FUNCTION_BLOCK C_BINARYREADER
VAR_INPUT
END_VAR
VAR_OUTPUT
END_VAR
VAR
	_BASESTREAM 	: I_STREAM;
END_VAR

PROPERTY BaseStream : I_STREAM
GET
BaseStream := _BASESTREAM;
END_GET
END_PROPERTY

METHOD Close : DINT
VAR_INPUT
END_VAR
Close := _BASESTREAM.Close();
_BASESTREAM := 0;
RETURN;
END_METHOD

METHOD New : DINT
VAR_INPUT
	STREAM : I_STREAM;
END_VAR
IF STREAM = 0 THEN
	New := 1;
	RETURN;
ELSE
	IF STREAM.IsValid THEN
		_BASESTREAM := STREAM;
		_BASESTREAM.Seek( 0, E_STREAMSEEKTYPE.Origin);
		New := -1;
		RETURN;
	ELSE
		New := 1;
		RETURN;
	END_IF
END_IF
END_METHOD

METHOD ReadBool : DINT
VAR_INPUT
	out_data : POINTER TO BOOL;
END_VAR
IF _BASESTREAM = 0 THEN
	ReadBool := 1;
	RETURN;
END_IF

ReadBool := _BASESTREAM.Read(out_data , 1);
RETURN;
END_METHOD

METHOD ReadBytes : DINT
VAR_INPUT
	out_data 	: POINTER TO BYTE;
	length		: UDINT;
END_VAR
IF _BASESTREAM = 0 THEN
	ReadBytes := 1;
	RETURN;
END_IF

ReadBytes := _BASESTREAM.Read(out_data, length);
RETURN;
END_METHOD

METHOD ReadDouble : DINT
VAR_INPUT
	out_data : POINTER TO LREAL;
END_VAR
IF _BASESTREAM = 0 THEN
	ReadDouble := 1;
	RETURN;
END_IF

ReadDouble := _BASESTREAM.Read(out_data , 8);
RETURN;
END_METHOD

METHOD ReadFloat : DINT
VAR_INPUT
	out_data : POINTER TO REAL;
END_VAR
IF _BASESTREAM = 0 THEN
	ReadFloat := 1;
	RETURN;
END_IF

ReadFloat := _BASESTREAM.Read(out_data , 4);
RETURN;
END_METHOD

METHOD ReadInt16 : DINT
VAR_INPUT
	out_data : POINTER TO INT;
END_VAR
IF _BASESTREAM = 0 THEN
	ReadInt16 := 1;
	RETURN;
END_IF

ReadInt16 := _BASESTREAM.Read(out_data , 2);
RETURN;
END_METHOD

METHOD ReadInt32 : DINT
VAR_INPUT
	out_data : POINTER TO DINT;
END_VAR
IF _BASESTREAM = 0 THEN
	ReadInt32 := 1;
	RETURN;
END_IF

ReadInt32 := _BASESTREAM.Read(out_data , 4);
RETURN;
END_METHOD

METHOD ReadString : DINT
VAR_INPUT
	out_data 	: PVOID;
	length		: UDINT;
END_VAR
IF _BASESTREAM = 0 THEN
	ReadString := 1;
	RETURN;
END_IF

ReadString := _BASESTREAM.Read(out_data, length);
RETURN;
END_METHOD

METHOD ReadUInt16 : DINT
VAR_INPUT
	out_data : POINTER TO UINT;
END_VAR
IF _BASESTREAM = 0 THEN
	ReadUInt16 := 1;
	RETURN;
END_IF

ReadUInt16 := _BASESTREAM.Read(out_data , 4);
RETURN;
END_METHOD

METHOD ReadUInt32 : DINT
VAR_INPUT
	out_data : POINTER TO UDINT;
END_VAR
IF _BASESTREAM = 0 THEN
	ReadUInt32 := 1;
	RETURN;
END_IF

ReadUInt32 := _BASESTREAM.Read(out_data , 4);
RETURN;
END_METHOD

METHOD Reset : DINT
VAR_INPUT
END_VAR
_BASESTREAM 	:= 0;
Reset := -1;
END_METHOD

END_FUNCTION_BLOCK

(* stored: Version 1.1.0.1, ProductVersion 3.1.4019.2
   POU C_BINARYREADER: Id {3b66d005-3f47-4af4-a375-894516dc8bea}, SpecialFunc None
   Property BaseStream: Id {71cc1926-e2dc-417b-be5f-3e2a654df2aa}
   Get Get: Id {e0c76d2d-5cef-40c9-82e4-8af46b1fce9d}
   Method Close: Id {de3cb16b-5206-41f8-a6b6-71c7bc0eb741}
   Method New: Id {4608d601-859c-47f4-831c-e01655b347f4}
   Method ReadBool: Id {76d45542-60ae-421d-a421-b25cd500e521}
   Method ReadBytes: Id {369d9618-2206-40c5-ad7f-cfb8812abbed}
   Method ReadDouble: Id {db11d57f-7dd3-4a73-85f8-532f0941f54f}
   Method ReadFloat: Id {44748d10-e06c-4cd0-983b-1dae6ee03d82}
   Method ReadInt16: Id {2b50ad5d-6d0a-4a08-a27e-1dee1b4acca2}
   Method ReadInt32: Id {555c708b-06af-4983-bc95-ad72bfff7519}
   Method ReadString: Id {8bbb68ff-c92f-4a55-8401-1cce0167fdf4}
   Method ReadUInt16: Id {73cf70b9-22f9-426b-a7d1-458ae4cb6acc}
   Method ReadUInt32: Id {b9ecc356-b187-4340-98f9-de3663fa31b7}
   Method Reset: Id {385790db-108f-4dd3-919c-3cd67536efd8} *)
